{attribute 'qualified_only'}
{attribute 'strict'}
TYPE CONTROL :
(
	StartConveyor := 0000_0001,
	StopConveyor := 0000_0000
) BYTE;
END_TYPE

(* stored: Version 1.1.0.1, ProductVersion 3.1.4024.9
   DUT CONTROL: Id {4bc6e21b-e756-48a1-99e1-c9583bbb536e} *)
